Staubli VAL3: stop.pgx

program stop()
begin
  //header begin
  //  PROGRAM STOP()
  //    peforms orderly shutdown functions
  //
  // initial release KN
  //header end
  //
  userPage()
  title(" SHUT DOWN ")
  cls()
  gotoxy(0,4)
  putln("WAITING:  Disabling Arm Power...")
  stopMove()
  resetMotion()
  disablePower()
  wait(isPowered()==false)
  //
  // stop tasks
  taskKill("MonitorZone")
  taskKill("RemoteControl")
  taskKill("MonitorHalt")
  taskKill("RemoteMotion")
  taskKill("iocCmdHandler")
  taskKill("RemoteMotion")
  taskKill("SimESTOP")
  //
  // tell user to press the MENU button to return to Application Menu
  cls()
  title(">>  PROGRAM STOPPED <<")
  gotoxy(0,2)
  put("Use MENU Button to return")
  gotoxy(0,3)
  put("to Main VAL3 Application Menu")
  //
  //done
end
